Yaskawa INFORM job: VALVE4.JBI

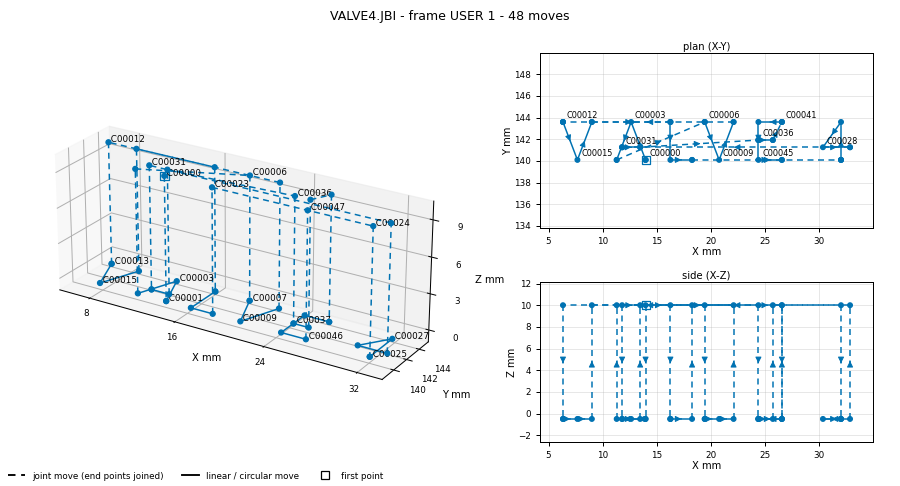
[picture p0: tool path of VALVE4.JBI in frame USER 1, 48 of 48 moves have a stored position in this frame; points joined in program order, loops and branches not executed]
/JOB
//NAME VALVE4
//POS
///NPOS 48,0,0,0,0,0
///USER 1
///TOOL 0
///POSTYPE USER
///RECTAN
///RCONF 1,0,0,0,0,0,0,0,0,0,0,0,0,0,0,0,0,0,0,0,0,0,0,0
C00000=13.956,140.101,10.000,0.0000,0.0000,0.0000
C00001=13.956,140.101,-0.500,0.0000,0.0000,0.0000
C00002=13.956,140.101,-0.500,0.0000,0.0000,0.0000
C00003=12.623,143.601,-0.500,0.0000,0.0000,0.0000
C00004=11.290,140.101,-0.500,0.0000,0.0000,0.0000
C00005=11.290,140.101,10.000,0.0000,0.0000,0.0000
C00006=19.415,143.601,10.000,0.0000,0.0000,0.0000
C00007=19.415,143.601,-0.500,0.0000,0.0000,0.0000
C00008=19.415,143.601,-0.500,0.0000,0.0000,0.0000
C00009=20.748,140.101,-0.500,0.0000,0.0000,0.0000
C00010=22.081,143.601,-0.500,0.0000,0.0000,0.0000
C00011=22.081,143.601,10.000,0.0000,0.0000,0.0000
C00012=6.331,143.601,10.000,0.0000,0.0000,0.0000
C00013=6.331,143.601,-0.500,0.0000,0.0000,0.0000
C00014=6.331,143.601,-0.500,0.0000,0.0000,0.0000
C00015=7.665,140.101,-0.500,0.0000,0.0000,0.0000
C00016=8.998,143.601,-0.500,0.0000,0.0000,0.0000
C00017=8.998,143.601,10.000,0.0000,0.0000,0.0000
C00018=16.248,143.601,10.000,0.0000,0.0000,0.0000
C00019=16.248,143.601,-0.500,0.0000,0.0000,0.0000
C00020=16.248,143.601,-0.500,0.0000,0.0000,0.0000
C00021=16.248,140.101,-0.500,0.0000,0.0000,0.0000
C00022=18.248,140.101,-0.500,0.0000,0.0000,0.0000
C00023=18.248,140.101,10.000,0.0000,0.0000,0.0000
C00024=31.998,140.101,10.000,0.0000,0.0000,0.0000
C00025=31.998,140.101,-0.500,0.0000,0.0000,0.0000
C00026=31.998,140.101,-0.500,0.0000,0.0000,0.0000
C00027=31.998,143.601,-0.500,0.0000,0.0000,0.0000
C00028=30.331,141.268,-0.500,0.0000,0.0000,0.0000
C00029=32.831,141.268,-0.500,0.0000,0.0000,0.0000
C00030=32.831,141.268,10.000,0.0000,0.0000,0.0000
C00031=11.790,141.268,10.000,0.0000,0.0000,0.0000
C00032=11.790,141.268,-0.500,0.0000,0.0000,0.0000
C00033=11.790,141.268,-0.500,0.0000,0.0000,0.0000
C00034=13.456,141.268,-0.500,0.0000,0.0000,0.0000
C00035=13.456,141.268,10.000,0.0000,0.0000,0.0000
C00036=24.373,141.934,10.000,0.0000,0.0000,0.0000
C00037=24.373,141.934,-0.500,0.0000,0.0000,0.0000
C00038=24.373,141.934,-0.500,0.0000,0.0000,0.0000
C00039=25.706,141.934,-0.500,0.0000,0.0000,0.0000
C00040=25.706,141.934,10.000,0.0000,0.0000,0.0000
C00041=26.540,143.601,10.000,0.0000,0.0000,0.0000
C00042=26.540,143.601,-0.500,0.0000,0.0000,0.0000
C00043=26.540,143.601,-0.500,0.0000,0.0000,0.0000
C00044=24.373,143.601,-0.500,0.0000,0.0000,0.0000
C00045=24.373,140.101,-0.500,0.0000,0.0000,0.0000
C00046=26.540,140.101,-0.500,0.0000,0.0000,0.0000
C00047=26.540,140.101,10.000,0.0000,0.0000,0.0000
//INST
///DATE 2025/08/05 10:19
///ATTR SC,RW,RJ
////FRAME USER 1
///GROUP1 RB1
NOP
DOUT OT#(1) OFF
DOUT OT#(1) OFF
TIMER T=1.000
MOVJ C00000 VJ=10.00
MOVJ C00001 VJ=10.00
DOUT OT#(1) ON
TIMER T=1.000
MOVL C00002 V=1.0 PL=0
MOVL C00003 V=1.0 PL=0
MOVL C00004 V=1.0 PL=0
DOUT OT#(1) OFF
TIMER T=1.000
MOVJ C00005 VJ=10.00
MOVJ C00006 VJ=10.00
MOVJ C00007 VJ=10.00
DOUT OT#(1) ON
TIMER T=1.000
MOVL C00008 V=1.0 PL=0
MOVL C00009 V=1.0 PL=0
MOVL C00010 V=1.0 PL=0
DOUT OT#(1) OFF
TIMER T=1.000
MOVJ C00011 VJ=10.00
MOVJ C00012 VJ=10.00
MOVJ C00013 VJ=10.00
DOUT OT#(1) ON
TIMER T=1.000
MOVL C00014 V=1.0 PL=0
MOVL C00015 V=1.0 PL=0
MOVL C00016 V=1.0 PL=0
DOUT OT#(1) OFF
TIMER T=1.000
MOVJ C00017 VJ=10.00
MOVJ C00018 VJ=10.00
MOVJ C00019 VJ=10.00
DOUT OT#(1) ON
TIMER T=1.000
MOVL C00020 V=1.0 PL=0
MOVL C00021 V=1.0 PL=0
MOVL C00022 V=1.0 PL=0
DOUT OT#(1) OFF
TIMER T=1.000
MOVJ C00023 VJ=10.00
MOVJ C00024 VJ=10.00
MOVJ C00025 VJ=10.00
DOUT OT#(1) ON
TIMER T=1.000
MOVL C00026 V=1.0 PL=0
MOVL C00027 V=1.0 PL=0
MOVL C00028 V=1.0 PL=0
MOVL C00029 V=1.0 PL=0
DOUT OT#(1) OFF
TIMER T=1.000
MOVJ C00030 VJ=10.00
MOVJ C00031 VJ=10.00
MOVJ C00032 VJ=10.00
DOUT OT#(1) ON
TIMER T=1.000
MOVL C00033 V=1.0 PL=0
MOVL C00034 V=1.0 PL=0
DOUT OT#(1) OFF
TIMER T=1.000
MOVJ C00035 VJ=10.00
MOVJ C00036 VJ=10.00
MOVJ C00037 VJ=10.00
DOUT OT#(1) ON
TIMER T=1.000
MOVL C00038 V=1.0 PL=0
MOVL C00039 V=1.0 PL=0
DOUT OT#(1) OFF
TIMER T=1.000
MOVJ C00040 VJ=10.00
MOVJ C00041 VJ=10.00
MOVJ C00042 VJ=10.00
DOUT OT#(1) ON
TIMER T=1.000
MOVL C00043 V=1.0 PL=0
MOVL C00044 V=1.0 PL=0
MOVL C00045 V=1.0 PL=0
MOVL C00046 V=1.0 PL=0
DOUT OT#(1) OFF
TIMER T=1.000
MOVJ C00047 VJ=10.00
DOUT OT#(1) OFF
END
